FUNCTION_BLOCK T_NumberCommandTask_1 EXTENDS T_MockCommandTask IMPLEMENTS I_NumberResultTask
VAR
  _result : LREAL;
END_VAR

PROPERTY Result : LREAL
GET
Result := _result;
END_GET
END_PROPERTY

METHOD PUBLIC SetResultValue
VAR_INPUT
  value : LREAL;
END_VAR
_result := value;
END_METHOD

END_FUNCTION_BLOCK

(* stored: Version 1.1.0.1
   POU T_NumberCommandTask_1: Id {8342416d-e60b-4957-8e0f-8456f67af4e5}, SpecialFunc None
   Property Result: Id {7e8a2101-fe46-4137-aa9f-a1b31710014a}
   Get Get: Id {1fb92c21-dd6a-4f6d-85e5-3a84b816d3bb}
   Method SetResultValue: Id {5d427fa2-6314-4a40-a856-79cdedeb2fc4} *)
